(* CODESYS project TestOSCAT.project

Project tree, tasks and I/O mapping:
  Device : OWEN PLC323.03-CS1.WEB, Owen, order no. 005, version 3.5.0.40
      unmapped channels: Discrete Outputs, Discrete inputs
    application Application
      libraries: NETWORK, 1.2.1.0 (OSCAT); BASIC, 3.31 (OSCAT); SysSocket23, 3.4.1.0 (System)
      task MainTask (cyclic, interval t#20ms, priority 1, watchdog 2000 ms x 1) calls PLC_PRG
      program PLC_PRG [ST]
      SOCKET/
        function block SOCKET_SERVER [ST]
        function block IP_CONTROL2_1 [ST]
        program NETWORK [ST]
      Message/
        function extractPayload [ST]
        function getMask [ST]
        function getOpcode [ST]
        function getPayloadLength [ST]
        function isFin [ST]
        function isMasked [ST]
        function sendPacket [ST]
      private/
        function byteArrayToString [ST]
        function sendError [ST]
        function sendResponse [ST]
        function StringToByteArray [ST]
        function block HttpHeader [ST]
      global variables GVL
    Owen:Internal
        unmapped channels: Discrete Outputs, Discrete inputs
*)

// Device/Application/GVL
VAR_GLOBAL
	MAX_RECEIVE_TCP_SERVER 	:UDINT := 512;
	MAX_SEND_TCP_SERVER 	:UDINT := 512;
END_VAR

// Device/Application/PLC_PRG
PROGRAM PLC_PRG
VAR
	S_BUF_WEB: OSCAT_NETWORK.NETWORK_BUFFER_SHORT;
	R_BUF_WEB: OSCAT_NETWORK.NETWORK_BUFFER_SHORT;
	counter: INT;
END_VAR
VAR CONSTANT
	CLOSED 			:	BYTE := 0;
	OPEN 			:	BYTE := 1;
END_VAR

NETWORK(S_BUF_WEB := S_BUF_WEB, R_BUF_WEB := R_BUF_WEB);

IF NETWORK.state = OPEN THEN

counter := counter + 1;

	IF (counter > 300) THEN
	
		S_BUF_WEB.BUFFER[0] := 6;
		S_BUF_WEB.BUFFER[1] := 2;
		S_BUF_WEB.BUFFER[2] := 3;
		S_BUF_WEB.BUFFER[3] := 4;
		S_BUF_WEB.SIZE 		:= 4;
	
		counter := 0;
	
	END_IF

ELSE
		counter := 0;
END_IF

END_PROGRAM

// Device/Application/SOCKET/NETWORK
PROGRAM NETWORK
VAR_IN_OUT
	S_BUF_WEB: OSCAT_NETWORK.NETWORK_BUFFER_SHORT;
	R_BUF_WEB: OSCAT_NETWORK.NETWORK_BUFFER_SHORT;
END_VAR
VAR

	IP_CONTROL2_0: IP_CONTROL2_1;
	S_SERVER_0: SOCKET_SERVER;
	
	IP_C: OSCAT_NETWORK.IP_C;
	S_BUF: OSCAT_NETWORK.NETWORK_BUFFER_SHORT;
	R_BUF: OSCAT_NETWORK.NETWORK_BUFFER_SHORT;
	
	
	
	DATA: ARRAY [0..255] OF WORD;
	
	Request:STRING(1024);	
	
	counter: INT;
	VMAP: ARRAY [1..10] OF  OSCAT_NETWORK.VMAP_DATA;
	
	
	(*Request		:	WebSocketRequest;*)
	HttpHeader_Web : HttpHeader;
	
	state: BYTE;
	i: INT;
	RequestValid: BOOL;
	Respons: POINTER TO STRING;
	b: BOOL;
	opcode: BYTE;
	payLen: DINT;
	ENABLE: BOOL;
END_VAR
VAR CONSTANT
	CLOSED 			:	BYTE := 0;
	OPEN 			:	BYTE := 1;
	SHAPost 		: 	STRING := '258EAFA5-E914-47DA-95CA-C5AB0DC85B11';
END_VAR



S_SERVER_0(IP_C := IP_C, S_BUF := S_BUF, R_BUF := R_BUF, ENABLE := ENABLE, UDP := FALSE);
IP_CONTROL2_0(IP_C := IP_C,S_BUF := S_BUF, R_BUF := R_BUF, IP := , PORT := 200, TIME_OUT :=T#10S);

IF IP_CONTROL2_0.CLOSED THEN state := CLOSED; END_IF
IF R_BUF_WEB.SIZE <> 0 THEN R_BUF_WEB.SIZE := 0; END_IF

IF NOT ENABLE AND IP_CONTROL2_0.CLOSED THEN ENABLE := TRUE; END_IF
(*
counter := counter + 1;

IF (counter > 300 AND IP_CONTROL2_0.OPEN) THEN

	S_BUF_WEB.BUFFER[0] := 6;
	S_BUF_WEB.BUFFER[1] := 2;
	S_BUF_WEB.BUFFER[2] := 3;
	S_BUF_WEB.BUFFER[3] := 4;
	S_BUF_WEB.SIZE 		:= 4;

	counter := 0;

END_IF

IF (counter > 300 AND IP_CONTROL2_0.CLOSED) THEN
	counter := 0;
END_IF
*)
IF state = CLOSED AND S_BUF.SIZE = UINT#0 AND R_BUF.SIZE >= UINT#1 THEN	(* Datensenden nicht aktiv und Daten wurden empfangen *)
			
			(*FOR i := 0 TO R_BUF.SIZE-1 DO
			S_BUF.BUFFER[i] := R_BUF.BUFFER[i];
			END_FOR
			S_BUF.SIZE := R_BUF.SIZE;*)
			
			HttpHeader_Web(arr := ADR(R_BUF.BUFFER));
			
			IF FINDB(HttpHeader_Web.Header[0], 'GET') <> 0 THEN RequestValid := TRUE; 
			ELSE
				 RequestValid := FALSE; 
			END_IF
			
			IF RequestValid THEN
				sendResponse(sendBuffer := ADR(S_BUF)+2, sendCount := ADR(S_BUF), HttpHeader_Web.Header);
				state := OPEN;
				Respons := ADR(S_BUF.BUFFER);
			ELSE
				sendError(sendBuffer := ADR(S_BUF)+2, sendCount := ADR(S_BUF));
				state := CLOSED;  
			END_IF
	 
END_IF;

IF state = OPEN AND S_BUF.SIZE = UINT#0 AND R_BUF.SIZE >= UINT#1 THEN
	opcode := getOpcode(ADR(R_BUF.BUFFER));
	payLen := getPayloadLength(ADR(R_BUF.BUFFER));
	
	IF (opcode = 2 AND R_BUF_WEB.SIZE = 0 AND isFin(ADR(R_BUF.BUFFER))) THEN
		extractPayload(ADR(R_BUF.BUFFER), ADR(R_BUF_WEB));
		
	ELSIF opcode = 8 THEN
		ENABLE := FALSE;
		state := CLOSED;
	END_IF
	
END_IF

IF state = OPEN AND S_BUF_WEB.SIZE > 0 THEN
		sendPacket(ADR(S_BUF), ADR(S_BUF_WEB));
	S_BUF_WEB.SIZE := 0;
END_IF


IF  state = OPEN AND S_BUF_WEB.SIZE > 0 THEN
	b := TRUE;
END_IF

END_PROGRAM

// Device/Application/private/sendResponse
FUNCTION sendResponse : BOOL
VAR_INPUT
	sendBuffer		:	POINTER TO ARRAY[0..1024] OF BYTE;
	sendCount		:	POINTER TO INT;
	Header			: 	ARRAY [0..20] OF STRING(255);
END_VAR
VAR CONSTANT
	SHAPost 			: 	STRING := '258EAFA5-E914-47DA-95CA-C5AB0DC85B11';
END_VAR
VAR
	sendSize		:	UINT;
	i					:	DINT;
	keyHeader			:	POINTER TO HttpHeader;
	key					:	STRING;
	
	abDigest			:	ARRAY[0..19] OF BYTE;
	conabDigest			:	ARRAY[0..20] OF BYTE;
	sDigest			:	STRING;

	abDigestBase64	:	ARRAY[0..32] OF BYTE;
	sDigestBase64	:	STRING;

	resp				:	ARRAY [0..5] OF STRING;
	b: BOOL;
	Done: BOOL;
	
	SHA1 : OSCAT_NETWORK.SHA1_STR;
	BASE64_ENCODE: OSCAT_NETWORK.BASE64_ENCODE_STR;
END_VAR

i := 0;

WHILE (FINDB(Header[i], 'Sec-WebSocket-Key') = 0) DO
	i := i + 1;
END_WHILE

Key := OSCAT_BASIC.Standard.MID(Header[i],24,FINDB(Header[i], ':')+2);
Key := OSCAT_BASIC.Standard.CONCAT(Key,SHAPost);

WHILE NOT SHA1.DONE DO
SHA1(Run := TRUE, str := Key, sha1 := abDigest); 
END_WHILE;

FOR i := 0 TO 19 DO
	conabDigest[i] := abDigest[i];
END_FOR

conabDigest[20] := 0;

sDigest := byteArrayToString(ADR(conabDigest));

WHILE NOT BASE64_ENCODE.DONE DO
BASE64_ENCODE(Run := TRUE, str1 := sDigest, str2 := sDigestBase64);
END_WHILE;



resp[0]:='HTTP/1.1 101 Switching Protocols';
resp[1]:='Upgrade: websocket';
resp[2]:='Connection: Upgrade';
resp[3]:=CONCAT('Sec-WebSocket-Accept: ', sDigestBase64);

sendSize := DINT_TO_UINT(StringToByteArray(sendBuffer, ADR(resp)));
sendCount^ := sendSize;
b := TRUE;

END_FUNCTION

// Device/Application/private/byteArrayToString
FUNCTION byteArrayToString : STRING(1024)
VAR_INPUT
	arr : POINTER TO ARRAY[0..1024] OF BYTE;
END_VAR
VAR
	p	: POINTER TO BYTE;
	str	: STRING (1024);
	i	: DINT := 0;
END_VAR

p := ADR(str);

WHILE (arr^[i] > 0) DO

  	p^ := arr^[i];
	i := i + 1;
	p := p + 1;

END_WHILE

p^ := 0;

byteArrayToString := str;

END_FUNCTION

// Device/Application/private/StringToByteArray
FUNCTION StringToByteArray : DINT
VAR_INPUT
	sendBuffer	:	POINTER TO ARRAY [0..1024] OF BYTE;
	str			:	POINTER TO ARRAY [0..5] OF STRING;
END_VAR
VAR
	p			:	POINTER TO BYTE;
	t			:	STRING;
	i,j			:	DINT;
END_VAR

i:=0; j:=0;
t := str^[0];

WHILE (LEN(t) > 0) DO

	p := ADR(str^[i]);
	WHILE (p^ > 0) DO
	 	sendBuffer^[j] := p^;
		j:=j + 1;
		p:=p+1;
	END_WHILE

	sendBuffer^[j] := 13;
	j := j + 1;
	sendBuffer^[j] := 10;
	j := j + 1;

	i := i + 1;
	t := str^[i];

END_WHILE

sendBuffer^[j] := 13;
j := j + 1;
sendBuffer^[j] := 10;
j := j + 1;


StringToByteArray := j;

END_FUNCTION

// Device/Application/private/HttpHeader
FUNCTION_BLOCK HttpHeader
VAR_INPUT
	arr : POINTER TO ARRAY[0..1024] OF BYTE;
END_VAR
VAR_OUTPUT
	Header	: ARRAY [0..20] OF STRING(255);
END_VAR
VAR
	p	: POINTER TO BYTE;
	str	: STRING (1024);
	i	: DINT := 0;

	j: INT;
END_VAR

j := 0;
i := 0;
p := ADR(Header[j]);

WHILE (arr^[i] > 0) DO

	
IF arr^[i-1] = 16#0D AND arr^[i] = 16#0A  THEN

p^ := arr^[i];
i := i + 1;
p := p + 1;
	
p^ := 0;
j := j + 1;
p := ADR(Header[j]);	
END_IF

 	p^ := arr^[i];
	i := i + 1;
	p := p + 1;
	
END_WHILE

END_FUNCTION_BLOCK

// Device/Application/private/sendError
FUNCTION sendError : BOOL
VAR_INPUT
	sendBuffer			:	POINTER TO ARRAY[0..1024] OF BYTE;
	sendCount			:	POINTER TO INT;
END_VAR
VAR
	resp					:	ARRAY [0..5] OF STRING;
	sendSize: UINT;
END_VAR

resp[0]:='HTTP/1.1 400 Bad Request';

sendSize := DINT_TO_UINT(StringToByteArray(sendBuffer, ADR(resp)));
sendCount^ := sendSize;

END_FUNCTION

// Device/Application/Message/getOpcode
FUNCTION getOpcode : BYTE
VAR_INPUT
	msg		:	POINTER TO ARRAY[0..1024] OF BYTE;
END_VAR
VAR
END_VAR

getOpcode.0 := msg^[0].0;
getOpcode.1 := msg^[0].1;
getOpcode.2 := msg^[0].2;
getOpcode.3 := msg^[0].3;

END_FUNCTION

// Device/Application/Message/getPayloadLength
FUNCTION getPayloadLength : DINT
VAR_INPUT
	msg		:	POINTER TO ARRAY[0..1024] OF BYTE;
END_VAR
VAR
	tmp		:	DINT;
	wordTmp	:	WORD;
END_VAR

tmp.0 := msg^[1].0;
tmp.1 := msg^[1].1;
tmp.2 := msg^[1].2;
tmp.3 := msg^[1].3;
tmp.4 := msg^[1].4;
tmp.5 := msg^[1].5;
tmp.6 := msg^[1].6;

IF (tmp = 127) THEN
	tmp := -1;
END_IF

IF (tmp = 126) THEN
	wordTmp := SHL(msg^[2], 8) + msg^[3];
	tmp := WORD_TO_DINT(wordTmp) ;
END_IF

getPayloadLength := tmp;

END_FUNCTION

// Device/Application/Message/isFin
FUNCTION isFin : BOOL
VAR_INPUT
	msg	:	POINTER TO ARRAY[0..1024] OF BYTE;
END_VAR
VAR
END_VAR

isFin := msg^[0].7;

END_FUNCTION

// Device/Application/Message/extractPayload
FUNCTION extractPayload : BOOL
VAR_INPUT
	pMsg		:	POINTER TO ARRAY[0..1024] OF BYTE;
	pPkt		:	POINTER TO OSCAT_NETWORK.NETWORK_BUFFER_SHORT;
END_VAR
VAR
	mask		:	ARRAY[0..3] OF BYTE;
	j			:	DINT := 0;
	payLen	:	DINT;
	i			:	DINT := 0;
END_VAR

payLen := getPayloadLength(pMsg);

IF (payLen > 125 OR payLen = -1) THEN
	extractPayload := FALSE;
	RETURN;
END_IF

pPkt^.SIZE := 0;
mask := getMask(pMsg);


WHILE ( i < payLen) DO

	pPkt^.BUFFER[i] := pMsg^[6 + i] XOR mask[j];

	pPkt^.SIZE := pPkt^.SIZE + 1;

	i:= i + 1;
	j := i MOD 4;
END_WHILE

END_FUNCTION

// Device/Application/Message/getMask
FUNCTION getMask : ARRAY[0..3] OF BYTE
VAR_INPUT
	pMsg		:	POINTER TO ARRAY[0..1024] OF BYTE;
END_VAR
VAR
END_VAR

IF (isMasked(pMsg)) THEN

	getMask[0] := pMsg^[2];
	getMask[1] := pMsg^[3];
	getMask[2] := pMsg^[4];
	getMask[3] := pMsg^[5];

END_IF

END_FUNCTION

// Device/Application/Message/isMasked
FUNCTION isMasked : BOOL
VAR_INPUT
	msg		:	POINTER TO ARRAY[0..1024] OF BYTE;
END_VAR
VAR
END_VAR

isMasked := msg^[1].7;

END_FUNCTION

// Device/Application/Message/sendPacket
FUNCTION sendPacket : BOOL
VAR_INPUT
	pMsg			:	POINTER TO OSCAT_NETWORK.NETWORK_BUFFER_SHORT;
	pPkt			:	POINTER TO OSCAT_NETWORK.NETWORK_BUFFER_SHORT;
END_VAR
VAR
	I				: 	INT;
END_VAR

IF (pPkt^.Size > 125) THEN
	sendPacket := FALSE;
	RETURN;
END_IF

pMsg^.BUFFER[0] :=2#10000010; (* set opcode to 2 and fin bit *)

pMsg^.BUFFER[1] := UINT_TO_BYTE(pPkt^.size);
pMsg^.BUFFER[1].7 := FALSE; (* mask bit set *)

(* no mask bit set, sending data unmasked *)
FOR I := 0 TO DINT_TO_INT(pPkt^.size) DO
	pMsg^.BUFFER[2 + i ] := pPkt^.BUFFER[i];
END_FOR

pMsg^.SIZE := pPkt^.size + 2;
sendPacket := TRUE;

END_FUNCTION

// Device/Application/SOCKET/IP_CONTROL2_1
FUNCTION_BLOCK IP_CONTROL2_1
VAR_IN_OUT
	IP_C : OSCAT_NETWORK.IP_C; (* IP_Control Verwaltungsstruktur *)
	S_BUF : OSCAT_NETWORK.NETWORK_BUFFER_SHORT; (* Externer Sendbuffer *)
	R_BUF : OSCAT_NETWORK.NETWORK_BUFFER_SHORT; (* Externer Receivebuffer *)
END_VAR
VAR_INPUT
	IP : DWORD; (* IP Adresse *)
	PORT : WORD; (* Port Nummer *)
	TIME_OUT : TIME; (* Ueberwachungszeit Connect / Send / Receive *)
END_VAR
VAR
	c_time : UDINT; (* CONNECT-Time (Zeit bei nicht vorhandener Verbindung) *)
	s_time : UDINT; (* SEND-Time    (Zeit seit letzten Datensenden) *)
	r_time : UDINT; (* RECEIVE-Time (Zeit seit letztem Datenempfang) *)

	c_enable : BOOL; (* Connect: freigabe *)
	c_ip : DWORD; (* Connect: aktuelle IP-Adresse *)
	c_port : WORD; (* Connect: aktuelle Port-Nummer *)
	c_mode : BYTE; (* Connect: aktueller Mode UDP/TCP...... *)
	c_status : BYTE; (* Connect: Status (Errorcode) *)
	c_ready : BOOL; (* Connect: Verbindung aufgebaut *)
	c_ready_old : BOOL; (* Connect: letzter Zustand von c_ready für Flankenauswertung *)
	c_select : BOOL; (* non blocking mode - abfrage über select durchführen *)
	c_fdWrite : SOCKET_FD_SET;
	c_Timeout : SOCKET_TIMEVAL;

	s_total : INT; (* Send: Gesamtanzahl Bytes zum senden *)
	s_cur_pos : INT; (* Send: aktuelle Sendeposition *)
	s_cur_size : INT; (* Send: aktuelle Sendegroesse *)
	s_max_size : INT; (* Send: maximale Telegrammlänge fuer Senden *)
	s_start : BOOL; (* Send: Sende modus aktivieren *)
	s_active : BOOL; (* Send: Daten senden ist aktiv *)
	s_req : BOOL; (* Send: Start Daten senden *)
	s_done : BOOL; (* Send: ohne Fehler beendet *)
	s_status : BYTE; (* Send: Status (Errorcodes) *)

	r_status : BYTE; (* Receive: Status (Errorcodes) *)
	r_count : INT; (* Receive: Anzahl empfangener Bytes *)
	r_offset : INT; (* Receive: aktuelle Position in externen Receivebuffer *)
	r_max_size : INT; (* Receive: groesse des externen Empfangbuffers*)

	new_connection : BOOL; (* Neue Verbindungsparameter vorhanden *)
	tx : DWORD; (* letzter zeitwert *)
	error_time : DWORD; (* aktueller Timeout-Wert *)

	state: BYTE; (* schrittmerker für connect *)
	server_socket : DINT:= OSCAT_NETWORK.SOCKET_INVALID;
	socket : DINT:= OSCAT_NETWORK.SOCKET_INVALID;
	sockaddr : SOCKADDRESS;
	sockaddr_size : DWORD;
	plc_841 : BOOL;
	plc_881 : BOOL;
	dint_true : DINT := 1;
	bytes_received : DINT;
	bytes_sent : DINT;
	udp_mode : BOOL;

	(*LOG_MSG : LOG_MSG;
	_debug_enable : BOOL := TRUE;
	debug_index : INT;
	debug_ID : INT;
	debug_lasterror : DWORD;
	debug_last_id : INT := 255;
	state_last: BYTE;*)

	Result_SysSockRecv: UDINT;
END_VAR

VAR_OUTPUT
	OPEN:BOOL;
	CLOSED:BOOL;
END_VAR

VAR CONSTANT
	STOP : BYTE := 0;
	TS_INIT: BYTE := 1;
	TS_OPEN : BYTE:= 2;
	UDP_INIT : BYTE:= 31;
	TC_INIT : BYTE:= 51;
	TC_CONNECT : BYTE:= 52;
	C_WAIT : BYTE:= 250;
	C_CLOSE : BYTE:= 251;
END_VAR

(* ---------------------- Debug-Message ----------------------------*)
(*IF _debug_enable THEN
	IF IP_C.FIFO.ID > BYTE#0 THEN (* nur wenn Teilnehmer ID's vorhanden sind *)
		debug_index := IP_C.FIFO.NR;
		debug_ID := BYTE_TO_INT(IP_C.FIFO.X[debug_index]);
	END_IF;
END_IF;*)
(* -----------------------------------------------------------------------------*)

(* read system time *)
tx := OSCAT_BASIC.T_PLC_MS();

OPEN := c_ready;
CLOSED := NOT OPEN;

IF IP_C.C_PORT = 0 THEN
	IP_C.C_PORT := PORT; (* uebergebenen PORT durch parametrierten PORT ersetzen *)
END_IF;
IF IP_C.C_IP = 0 AND IP_C.C_MODE < 4 THEN
	IP_C.C_IP := IP; (* uebergebene IP durch paramtrierte IP ersetzen *)
END_IF;

new_connection := c_ip <> IP_C.C_IP OR c_mode <> IP_C.C_MODE OR c_port <> IP_C.C_PORT; (* neue Verbindungs erwünscht ? *)
c_enable := IP_C.C_ENABLE AND NOT new_connection;

IF IP_C.C_ENABLE AND IP_C.ERROR = 0 AND state = STOP THEN (* Freigabe,kein Fehler,kein Socket offen *)
	c_ip   := IP_C.C_IP;
	c_mode := IP_C.C_MODE;
	c_port := IP_C.C_PORT;
	plc_841 := ADR(%MW0)=16#30000000; (*750-841*)
	plc_881 := ADR(%MW0)=16#20000000; (*750-881*)
	udp_mode := C_MODE.0; (* Mode 1,3,5 = udp *)

	error_time := TIME_TO_DWORD(MAX(T#200ms,TIME_OUT));
	IP_C.TIME_RESET := TRUE; (* Alle Timer ruecksetzen *)

	r_max_size := SIZEOF(R_BUF.BUFFER);
	s_max_size := SIZEOF(S_BUF.BUFFER);

	IF C_MODE.0 THEN (* Mode: 1,3,5 = UDP CLIENT/SERVER *)
		state := UDP_INIT;
	ELSIF C_MODE = 0 THEN (* Mode: 0 = TCP CLIENT *)
		state := TC_INIT;
	ELSE
		state := TS_INIT; (* Mode: 2,4 = TCP SERVER *)
	END_IF;

	(* ---------------------- Debug-Message ----------------------------*)
	(*IF _debug_enable THEN
		LOG_CL.NEW_MSG := 'IP_CON: MODE ~1 / IP ~2 / PORT ~3 /ID ~6';
		LOG_CL.PRINTF[1] := BYTE_TO_STRING(C_MODE);
		LOG_CL.PRINTF[2] := IP4_TO_STRING(c_ip);
		LOG_CL.PRINTF[3] := WORD_TO_STRING(c_port);
		LOG_CL.PRINTF[6] := INT_TO_STRING(debug_ID);
		LOG_MSG();
	END_IF;*)
	(* -----------------------------------------------------------------------------*)

END_IF;

(* ---------------------- Debug-Message ----------------------------*)
(*IF  _debug_enable THEN
	IF state <> state_last THEN
		LOG_CL.NEW_MSG := 'IP_STEP ~1 -IP_ID ~6';
		LOG_CL.PRINTF[1] := BYTE_TO_STRING(state);
		LOG_CL.PRINTF[6] := INT_TO_STRING(debug_ID);
		LOG_MSG();
		state_last := state;
	END_IF;
END_IF;*)
(* -----------------------------------------------------------------------------*)

IF IP_C.TIME_RESET THEN (* Alle Timer ruecksetzen *)
	IP_C.TIME_RESET := FALSE; (* Reset rücksetzen *)
	c_time := tx; (* Connect Timer ruecksetzen *)
	s_time := tx; (* Send Timer ruecksetzen *)
	r_time := tx; (* Receive Timer ruecksetzen *)

	c_status := BYTE#0; (* letzten Connect Fehler rücksetzen *)
	s_status := BYTE#0; (* letzten Send Fehler rücksetzen *)
	r_status := BYTE#0; (* letzten Receive Fehler rücksetzen *)
END_IF;

(* ---------------------------------------------- *)

CASE state OF

UDP_INIT: (* UDP_CLIENT + SERVER *)
	socket := SysSockCreate(SOCKET_AF_INET, SOCKET_DGRAM, SOCKET_IPPROTO_IP);
	IF socket < 0 THEN
		c_status := 1; (* SysSockCreate failed *)
		state := C_CLOSE;
	ELSE
		SysSockSetOption(socket, SOCKET_SOL, SOCKET_SO_BROADCAST, ADR(dint_true), SIZEOF(dint_true)); (* allow broadcast *)
		SysSockIoctl(socket, SOCKET_FIONBIO, ADR(dint_true)); (* put socket in non-blocking mode *)
		sockaddr.sin_family := SOCKET_AF_INET;
		sockaddr.sin_port := SysSockHtons(c_port);
		sockaddr.sin_addr := SEL(c_mode = 1, SOCKET_INADDR_ANY, SysSockNtohl(c_ip));

		IF c_mode >= 2 THEN (* SERVER Mode *)
			IF SysSockBind(socket, ADR(sockaddr), SIZEOF(sockaddr)) THEN
				c_ready := TRUE; (* Connected *)
				state:= C_WAIT;
			ELSE
				c_status := 2; (* SysSockBind failed *)
				state := C_CLOSE;
			END_IF;
		ELSE
			c_ready := TRUE; (* Connected *)
			state:= C_WAIT;
		END_IF;
	END_IF;

(* ---------------------------------------------- *)

TC_INIT: (* TCP-CLIENT (AKTIV) *)
	socket := SysSockCreate(SOCKET_AF_INET, SOCKET_STREAM, SOCKET_IPPROTO_IP);
	IF socket < 0 THEN
		c_status := 1;  (* SysSockCreate failed *)
		state := C_CLOSE;
	ELSE
		IF plc_841 OR plc_881 THEN
			SysSockSetOption(socket,6,SOCKET_TCP_NODELAY, ADR(dint_true), SIZEOF(dint_true)); (* Set Push-Bit *)
		END_IF;
		SysSockIoctl(socket, SOCKET_FIONBIO, ADR(dint_true)); (* NonBlocking mode *)
		sockaddr.sin_family := SOCKET_AF_INET;
		sockaddr.sin_port := SysSockNtohs(c_port);
		sockaddr.sin_addr := SysSockNtohl(c_ip);
		c_select := FALSE;
		state := TC_CONNECT;
	END_IF;

(* ---------------------------------------------- *)

TC_CONNECT:
	IF NOT c_enable OR c_status = 255 THEN (* keine freigabe oder connect timeout *)
			state:= C_CLOSE;
	ELSE
		IF c_select = FALSE THEN
			IF SysSockConnect(socket,ADR(sockaddr),SIZEOF(sockaddr)) THEN
				c_ready := TRUE; (* Connected *)
				state:= C_WAIT;
			ELSE
				(* Connect durchgeführt, aber noch nicht verbunden, dann optional mit select-abfrage weitermachen *)
				c_select := OSCAT_NETWORK.SYSLIBSOCKETS_OPTION.0; (* Bit 0 = TCP-Client - use SysSockselect *)
			END_IF;
		ELSE
			c_Timeout.tv_sec := 0;
			c_Timeout.tv_usec := 0;
			c_fdWrite.fd_count := 1;
			c_fdWrite.fd_array[0] := socket;
			IF SysSockSelect(SOCKET_FD_SETSIZE,0,ADR(c_fdWrite),0, ADR(c_Timeout)) > 0 THEN
				c_ready := TRUE; (* Connected *)
				state:= C_WAIT;
			END_IF;
		END_IF;
	END_IF;

(* ---------------------------------------------- *)

TS_INIT: (* TCP-SERVER (PASSIV) *)
	server_socket := SysSockCreate(SOCKET_AF_INET, SOCKET_STREAM, SOCKET_IPPROTO_IP); (* Create Socket *)
	IF server_socket = SOCKET_INVALID THEN
		c_status := 1; (* SysSockCreate failed *)
		state:= C_CLOSE;
	ELSE (* Address bindings *)
		SysSockSetOption( server_socket, SOCKET_SOL, SOCKET_SO_REUSEADDR, ADR(dint_true), SIZEOF(dint_true) );
		sockaddr.sin_family:= SOCKET_AF_INET;
		sockaddr.sin_port := SysSockHtons(c_port);
		sockaddr.sin_addr := SOCKET_INADDR_ANY;
		IF NOT SysSockBind(server_socket, ADR(sockaddr), SIZEOF(sockaddr)) THEN
			c_status := 2; (* SysSockBind failed *)
			state := C_CLOSE;
		ELSIF NOT SysSockListen(server_socket, 1) THEN (* erzeugt Warteschlange für eine Verbindung *)
			c_status := 3; (* SysSockListen failed *)
			state:= C_CLOSE;
		ELSE
			SysSockIoctl(server_socket, SOCKET_FIONBIO, ADR(dint_true)); (* NonBlocking mode *)
			state:= TS_OPEN;
		END_IF;
	END_IF;

(* ---------------------------------------------- *)

TS_OPEN: (* Waiting for incomming connection *)
	sockaddr_size := SIZEOF(sockaddr);
	socket := SysSockAccept(server_socket, ADR(sockaddr), ADR(sockaddr_size));

	IF socket <> SOCKET_INVALID THEN (* neuer Verbindungswunsch vorhanden *)
		IF c_mode = BYTE#2 AND sockaddr.sin_addr <> SysSockNtohl(c_ip) THEN (* Mode 2 = TCP + PASSIVE + PORT + IP  auf richtige Partner-IP prüfen *)
			state:= C_CLOSE;
		ELSE
			IF plc_841 OR plc_881 THEN
				SysSockSetOption(socket, 6, SOCKET_TCP_NODELAY, ADR(dint_true), SIZEOF(dint_true)); (* Set Push-Bit *)
			END_IF;
			SysSockIoctl(socket, SOCKET_FIONBIO, ADR(dint_true)); (* NonBlocking mode *)
			c_ready := TRUE; (* Connected *)
			state := C_WAIT;
		END_IF;
	ELSIF NOT c_enable THEN (* keine freigabe mehr ? *)
			state:= C_CLOSE;
	END_IF;

(* ---------------------------------------------- *)

C_WAIT: (* Warten auf Anforderung für Beenden *)
	IF NOT c_enable OR NOT c_ready THEN
		state:= C_CLOSE;
	END_IF

(* ---------------------------------------------- *)

C_CLOSE: (* Close the Sockets *)
	c_ready := FALSE;
	IF socket >= 0 THEN
		IF (NOT plc_841) AND (NOT plc_881) THEN
			SysSockShutdown(socket, 0); (* 870 *)
		END_IF;
		SysSockClose(socket);
		socket := SOCKET_INVALID;
	END_IF
	IF server_socket >= 0 THEN
		IF (NOT plc_841) AND (NOT plc_881) THEN
			SysSockShutdown(server_socket, 0); (* 870 *)
		END_IF;
		SysSockClose(server_socket);
		server_socket := SOCKET_INVALID;
	END_IF
	state:= STOP;
END_CASE;

(* ---------------------------------------------- *)

IF c_ready THEN
	IF NOT c_ready_old THEN (* Verbindung aufgebaut - positive Flanke erkannt *)
		IP_C.C_STATE := 254;
		IP_C.TIME_RESET := TRUE; (* Alle Timer ruecksetzen *)
		(* ---------------------- Debug-Message ----------------------------*)
		(*IF _debug_enable THEN
			LOG_CL.NEW_MSG := 'IP_CON: CONNECTED -IP_ID ~6';
			LOG_CL.PRINTF[6] := INT_TO_STRING(debug_ID);
			LOG_MSG();
		END_IF;*)
		(* -----------------------------------------------------------------------------*)
	ELSE
		IP_C.C_STATE := 255; (* Verbindung ist aufgebaut *)
	END_IF;
ELSE
	IF c_ready_old THEN (* Verbindung abgebaut - negative Flanke erkannt *)
		IP_C.C_STATE := 1;
		IP_C.MAILBOX[1] := 0; (* Receive Info rücksetzen *)
		IP_C.MAILBOX[2] := 0; (* Send-Pause rücksetzen *)
		IP_C.MAILBOX[3] := 0; (* Receive-Pause rücksetzen *)
		IF NOT new_connection THEN
			s_active := FALSE; (* Sendeaktivitäten stoppen *)
			s_req := FALSE; (* Sendefreigabe rücksetzen *)
			S_BUF.SIZE := 0; (* Sendelänge löschen *)
			(* IP_C.TIME_RESET := TRUE; *) (* Alle Timer ruecksetzen *)
		END_IF;
		(* ---------------------- Debug-Message ----------------------------*)
		(*IF _debug_enable THEN
			LOG_CL.NEW_MSG := 'IP_CON: DISCONNECTED';
			LOG_MSG();
		END_IF;*)
		(* -----------------------------------------------------------------------------*)
	ELSE
		IP_C.C_STATE := 0; (* Verbindung ist abgebaut *)
	END_IF;
END_IF;

c_ready_old := c_ready;

(* Der Datenempfang wird angehalten solange ein Sendevorgang läuft *)
(* sonst kann es vorkommen das die Antwort-daten schon empfangen werden, *)
(* bevor der Sendevorgang vom programm abgeschlossen wurde *)

IF c_ready AND NOT s_active AND IP_C.MAILBOX[3] = 0 THEN
	IF R_BUF.SIZE >= INT_TO_UINT(r_max_size) THEN
		R_BUF.SIZE := UINT#0;
		r_status := 254; (* Empfangsbuffer wegen Überlauf rückgesetzt *)
	END_IF;

	r_offset := SEL(udp_mode,UINT_TO_INT(R_BUF.SIZE),0);
	r_count := r_max_size - r_offset;

	IF udp_mode THEN
		bytes_received := SysSockRecvFrom(socket, ADR(R_BUF.BUFFER), r_count, 0, ADR(sockaddr), SIZEOF(sockaddr));

		IF c_mode = BYTE#3 AND sockaddr.sin_addr <> SysSockNtohl(c_ip) THEN (* Mode 3 = UDP + PASSIVE + PORT + IP  auf richtige Partner-IP prüfen *)
			bytes_received := 0;
			R_BUF.SIZE := UINT#0;
			sockaddr.sin_port := SysSockNtohs(c_port);
			sockaddr.sin_addr := SysSockNtohl(c_ip);
		END_IF;

	ELSE
		bytes_received := SysSockRecv30(hSocket := socket,pbyBuffer := ADR(R_BUF.BUFFER[r_offset]), diBufferSize := r_count, diFlags := 0, pResult:= ADR(Result_SysSockRecv));
	END_IF;

	(*UDP: IPC returns -1 if no data available or error occured,841 returns -1 if error occured and 0 if no data available*)
	CASE Result_SysSockRecv OF
	(*-2147483648..-1: ; (* No data available or error occured *)*)
	 529: IF NOT udp_mode THEN (* TCP-Mode: socket wurde von remote geschlossen *)
			c_status := 253;
			c_ready := FALSE;
		END_IF;
	ELSE (* daten wurden empfangen *)
  		r_time := tx; (* Receive Timer ruecksetzen *)
		R_BUF.SIZE := INT_TO_UINT(r_offset + DINT_TO_UINT(bytes_received)); (* aktuelle buffersize eintragen *)
		IP_C.MAILBOX[1] := IP_C.MAILBOX[1] + 1; (* Receive Info *)
		IF IP_C.MAILBOX[1] = 0 THEN IP_C.MAILBOX[1] := 1; END_IF;

		(* ---------------------- Debug-Message ----------------------------*)
		(*IF _debug_enable THEN
			LOG_CL.NEW_MSG := 'IP_REC DATA: POS: ~1 : SIZE: ~2 TOTAL ~3 -IP_ID ~6';
			LOG_CL.PRINTF[1] := INT_TO_STRING(r_offset);
			LOG_CL.PRINTF[2] := INT_TO_STRING(r_count);
			LOG_CL.PRINTF[3] := UINT_TO_STRING(R_BUF.SIZE);
			LOG_CL.PRINTF[6] := INT_TO_STRING(debug_ID);
			LOG_MSG();
		END_IF;*)
		(* -----------------------------------------------------------------------------*)

	END_CASE
END_IF;

(* ---------------------------------------------- *)

IF S_BUF.SIZE > 0 THEN
	IF c_ready AND c_enable THEN
		IF NOT s_active AND IP_C.MAILBOX[2] = 0 THEN
			(* Gesamtanzahl an Bytes limitieren und uebergeben *)
			s_total := LIMIT(0,UINT_TO_INT(S_BUF.SIZE),r_max_size);
			s_cur_pos  := 0;
			s_cur_size := 0;
			s_start := TRUE; (* Daten kopieren und senden anstossen *)
			s_active := TRUE; (* Sende-Betrieb aktivieren *)
			(* ---------------------- Debug-Message ----------------------------*)
			(*IF _debug_enable THEN
				LOG_CL.NEW_MSG := 'IP_SEN INIT: TOTAL: ~1 -IP_ID ~6';
				LOG_CL.PRINTF[1] := INT_TO_STRING(S_TOTAL);
				LOG_CL.PRINTF[6] := INT_TO_STRING(debug_ID);
				LOG_MSG();
			END_IF;*)
			(* -----------------------------------------------------------------------------*)
		END_IF;

		IF s_done OR s_start THEN (* Daten senden aktiv *)

			s_start := FALSE;
			s_cur_pos := s_cur_pos + s_cur_size; (* neue Sende-Datenposition bestimmen *)
			IF s_total > s_cur_pos THEN (* weitere Daten zum senden vorhanden ? *)
				s_cur_size := s_total - s_cur_pos;
				s_cur_size := LIMIT(0, s_cur_size, s_max_size); (* Telegrammlänge begrenzen *)

				(* ---------------------- Debug-Message ----------------------------*)
				(*IF _debug_enable THEN
					LOG_CL.NEW_MSG := 'IP_SEN DATA: POS: ~1 : SIZE: ~2 TOTAL ~3 -IP_ID ~6';
					LOG_CL.PRINTF[1] := INT_TO_STRING(S_CUR_POS);
					LOG_CL.PRINTF[2] := INT_TO_STRING(S_CUR_SIZE);
					LOG_CL.PRINTF[3] := INT_TO_STRING(S_TOTAL);
					LOG_CL.PRINTF[6] := INT_TO_STRING(debug_ID);
					LOG_MSG();
				END_IF;*)
				(* -----------------------------------------------------------------------------*)

				s_time := tx; (* Send Timer ruecksetzen *)
				r_time := tx; (* Receive Timer ruecksetzen *)
				s_req := TRUE;

			ELSE
				(* keine weitere Sendedaten vorhanden -> Senden beenden *)
				s_req := FALSE;
				s_active := FALSE;
				S_BUF.SIZE := 0;
				(* ---------------------- Debug-Message ----------------------------*)
				(*IF _debug_enable THEN
					LOG_CL.NEW_MSG := 'IP_SEN FINISH -IP_ID ~6';
					LOG_CL.PRINTF[6] := INT_TO_STRING(debug_ID);
					LOG_MSG();
				END_IF;*)
				(* -----------------------------------------------------------------------------*)
			END_IF;
		END_IF;
	END_IF;
END_IF;

IF s_req THEN
	s_done := FALSE;
	IF udp_mode THEN
		bytes_sent := SysSockSendTo(socket, ADR(S_BUF.BUFFER[s_cur_pos]), s_cur_size, 0, ADR(sockaddr), SIZEOF(sockaddr));
	ELSE
		bytes_sent := SysSockSend(socket, ADR(S_BUF.BUFFER[s_cur_pos]), s_cur_size, 0);
	END_IF;

	CASE bytes_sent OF
	-2147483648..-1:	; (* ERROR: Noch nicht bereit um Daten aufzunehmen -> nächsten Zyklus wieder probieren *)
	 0: IF NOT udp_mode THEN (* TCP-Mode: socket wurde von remote geschlossen *)
			c_status := 253;
			c_ready := FALSE;
		END_IF;
	ELSE
		s_done := TRUE;
		s_cur_size := DINT_TO_INT(bytes_sent); (* Anzahl der wirklich versendeten Bytes übernehmen *)
		(* ---------------------- Debug-Message ----------------------------*)
		(*IF _debug_enable THEN
			LOG_CL.NEW_MSG := 'IP_SEN SEND_COUNT ~1 -IP_ID ~6';
			LOG_CL.PRINTF[1] := DINT_TO_STRING(s_cur_size);
			LOG_CL.PRINTF[6] := INT_TO_STRING(debug_ID);
			LOG_MSG();
		END_IF;*)
		(* -----------------------------------------------------------------------------*)
	END_CASE
END_IF;

(* ---------------------------------------------- *)

IF IP_C.R_OBSERVE = FALSE OR s_active THEN
    r_time := tx;
END_IF;

IF c_status = 0 AND tx - c_time > error_time AND c_enable AND NOT c_ready AND c_mode < 2 THEN (* Connect Timeout *)
	c_status := 255; (* Timeout-Fehler ausgeben *)
END_IF;
IF s_status = 0 AND tx - s_time > error_time AND s_active THEN (* Send Timeout *)
	s_status := 255; (* Timeout-Fehler ausgeben *)
END_IF;
IF r_status = 0 AND tx - r_time > error_time AND c_ready AND IP_C.R_OBSERVE THEN (* Receive Timeout *)
	r_status := 255; (* Timeout-Fehler ausgeben *)
END_IF;

IP_C.ERROR := OSCAT_BASIC.DWORD_OF_BYTE(c_status,s_status,r_status,0);

(* ---------------------- Debug-Message ----------------------------*)
(*IF  _debug_enable THEN
	IF (IP_C.ERROR <> debug_lasterror) THEN
		LOG_CL.NEW_MSG := 'IP_ERROR ~1 -IP_ID ~6';
		LOG_CL.PRINTF[1] := DWORD_TO_STRING(IP_C.ERROR);
		LOG_CL.PRINTF[6] := INT_TO_STRING(debug_ID);
		LOG_MSG();

		debug_lasterror := IP_C.ERROR;
		debug_last_id := debug_ID;
	END_IF;
END_IF;*)
(* -----------------------------------------------------------------------------*)

(* revision history
ks	18. oct. 2008	rev 1.0
	original version
ks	05. jan. 2009	rev 1.1
	zusätzlichen Parameter "Port" hinzugefügt, und Code bei Verbindungsaufbau angepasst
ks	28. feb. 2009	rev 1.2
	connect code angepasst und verkürzung der zyklen bei Send
ks	20. oct. 2009	rev 1.3
	network_buffer basis 0
ks	06. dec. 2009	rev 1.4
	receive_count MAILBOX[1]
ks	10. nov. 2010	rev 1.5
	send_pause MAILBOX[2] and receive_pause MAILBOX[3] 
ks	07. feb. 2011	rev 1.6
	Fehlercode 253 bei Remote-Verbindungsabbruch 
ks	30. may. 2011	rev 1.7
	Fehler bei Empfangsüberwachung
ks	26. july. 2011	rev 1.8
	Error-Reset, diverse optimierungen 
ks	26. feb. 2012	rev 1.9
	Code-Optimierung für höhere kompatibilität
*)

END_FUNCTION_BLOCK

// Device/Application/SOCKET/SOCKET_SERVER
FUNCTION_BLOCK SOCKET_SERVER
VAR_IN_OUT
	IP_C : OSCAT_NETWORK.IP_C;
	S_BUF : OSCAT_NETWORK.NETWORK_BUFFER_SHORT;
	R_BUF : OSCAT_NETWORK.NETWORK_BUFFER_SHORT;
(*	VMAP : ARRAY [1..10] OF OSCAT_NETWORK.VMAP_DATA;
	DATA : ARRAY [0..255] OF WORD;
*)
END_VAR
VAR_INPUT
(*	DATA_SIZE : INT;*)
	ENABLE : BOOL;
	UDP : BOOL;
END_VAR
VAR_OUTPUT
	ERROR : DWORD;
END_VAR
VAR
	MB_VMAP : OSCAT_NETWORK.MB_VMAP;
	adr1 : INT;
	adr2 : INT;
	points : INT;
	points2 : INT;
	coils : BYTE;
	mask : BYTE;
	idx1 : INT;
	idx2 : INT;
	bit_pos : INT;
	count : INT;
	fc : INT;
	i : INT;
	state : INT;
	ip_state : BYTE;
	ip_id : BYTE;
	IP_FIFO : OSCAT_NETWORK.IP_FIFO;
	w_tmp : WORD;
	last_cycle : TIME;
	tx : TIME;
	t : OSCAT_BASIC.TON;
	ip_error : BOOL;
END_VAR

(* read system time *)
tx := DWORD_TO_TIME(OSCAT_BASIC.T_PLC_MS());

(*
FOR i := 1 TO 10 DO
	IF VMAP[i].TIME_OUT > T#0s THEN
		VMAP[i].TIME_OUT := VMAP[i].TIME_OUT + tx - last_cycle;
	END_IF;
END_FOR;
*)

last_cycle := tx;
ip_error := IP_C.ERROR > DWORD#0;
IP_C.C_ENABLE := ENABLE;

CASE state OF
00: (* Warten auf Freigabe *)
	IF ENABLE THEN
		state := 10;
		ip_state := BYTE#1; (* Anmelden *)
	END_IF;

10: (* Bei IP_Control anmelden und auf freigabe warten *)
	IF ip_state = BYTE#3 THEN

		(* IP Datenverkehr einrichten *)
		IP_C.C_PORT := WORD#0; (* Port von IP_CONTROL verwenden *)
		IP_C.C_IP := DWORD#0; (* IP von IP_CONTROL verwenden *)
		IP_C.C_MODE := SEL(UDP,BYTE#4,BYTE#5); (* Mode: 4=TCP+PASSIV+PORT , 5=UDP+PASSIV+PORT *)
		IP_C.TIME_RESET := TRUE; (* Zeitueberwachung rücksetzen *)
		IP_C.C_ENABLE := ENABLE; (* Verbindungsaufbau freigeben *)
		IP_C.R_OBSERVE := FALSE; (* keine Empfangsueberwachung *)
		state := 20;
	END_IF;

20:	IF NOT ip_error THEN
		IF S_BUF.SIZE = UINT#0 AND R_BUF.SIZE >= UINT#1 THEN	(* Datensenden nicht aktiv und Daten wurden empfangen *)
			(*
			FOR i := 0 TO R_BUF.SIZE-1 DO
			S_BUF.BUFFER[i] := R_BUF.BUFFER[i];
			END_FOR
			S_BUF.SIZE := R_BUF.SIZE;
			*)
		END_IF;
	ELSE
		ERROR := IP_C.ERROR;
	END_IF;

	t(IN:= ip_error, PT:=T#5s);
	IF t.Q THEN
		IP_C.TIME_RESET := TRUE; (* Error Reset *)
	END_IF;



	R_BUF.SIZE := UINT#0; (* Empfangsdaten zerstören *)

	IF ENABLE = FALSE THEN
	    ip_state := BYTE#4; (* Abmelden *)
		state := 00;
	END_IF;
END_CASE;

(* IP_FIFO *)
IP_FIFO(FIFO:=IP_C.FIFO,STATE:=ip_state,ID:=ip_id);

END_FUNCTION_BLOCK
